// TIA Portal V18 export
DATA_BLOCK "ACC_AccessControl_idb"   // DB12
VERSION : 0.1
// stored: AutoNumber true, DBAccessibleFromOPCUA true, InstanceOfName AccessControl, InstanceOfType FB
"AccessControl"
   // VAR_INPUT
   //    SearchStatus : Int;
   //    RunArea : Bool;
   //    ACC_Ready : Bool;
   //    ACC_Run : Bool;
   //    ACC_StopBeam : Bool;
   //    Key : Bool;
   //    keyControl : Bool;
   //    Interlock : Bool;
   //    DoseAttenuation_Time : Time;
   //    StartAlarm_Time : Time;
   // END_VAR
   // VAR_OUTPUT
   //    StartAlarm : Bool;
   //    NoEntry : Bool;
   //    RestrictedEntry : Bool;
   //    ControlEntry : Bool;
   // END_VAR
   // VAR_IN_OUT
   //    AreaReady : Bool;
   //    BeamAllowed : Bool;
   // END_VAR
   // VAR
   //    State : Int;
   //    DoseAttenuation_Timer { S7_SetPoint := 'True'} : TON_TIME;
   //    StartAlarm_Timer { S7_SetPoint := 'True'} : TON_TIME;
   // END_VAR
BEGIN
END_DATA_BLOCK
